Fanuc KAREL source: kt00060.KL

-- PROVISIONAL review KL for V940-1; original PC SHA256 1cb13336a32c3d72ca695b3430573ebc0f6a524cb1e94895d5cea25c975ca418
-- Incomplete behavior may be omitted. Consult companion uncertainty JSON. Do not deploy.
PROGRAM KT00060
%NOLOCKGROUP
VAR
  R2 : REAL
  OUT : REAL
-- UNRESOLVED_DECL H1 type=002017
BEGIN
  -- V9_ZERO_TABLE_METADATA_HINT layout=0001; no indexed target words; source/name/runtime held
  -- UNRESOLVED_PC offsets 5-19; opcodes 2E,22,9D,33,B4
  -- UNRESOLVED_PC offsets 24-35; opcodes 2E,23
  -- UNRESOLVED_PC offsets 40-65; opcodes 22,9D,33,B3,21,29,64,29,6A,23
  -- UNRESOLVED_PC offsets 70-74; opcodes 7F
END KT00060
